{attribute 'OPC.UA.DA' := '0'}
TYPE SerialCommunication :
STRUCT
	Port : STRING;
	BaudRate : UDINT;
	DataFrame : STRING;
	FlowControl : SerialFlowControl;
	CanOverEthercat : CanOverEthercat;
END_STRUCT
END_TYPE

(* stored: Version 1.1.0.1, ProductVersion 3.1.4024.3
   DUT SerialCommunication: Id {328e7796-fb79-471e-ab76-fbc37a867be7} *)
